# EPICS IOC start-up script: iocBoot/common/startup.RK_CA3900.iocsh
# IOC shell script for R&K CA3900 SSA
# Includes modbus config and db loading
# Required macros:
# PORT - asyn port
# P - PV name prefix
# IP - IP address or host name

# Use the following commands for TCP/IP
# drvAsynIPPortConfigure(const char *portName, const char *hostInfo,
# 			 unsigned int priority, int noAutoConnect,
#			 int noProcessEos);

drvAsynIPPortConfigure("$(PORT)", "$(IP):502", 0,0,1)
dbLoadRecords("db/asynRecord.db","P=$(P), R=ASYN, PORT=$(PORT), ADDR=0,IMAX=0,OMAX=0")

# modbusInterposeConfig(const char *portName, modbusLinkType linkType,
#			int timeoutMsec, int writeDelayMsec)
# linkType 0 = TCP/IP
modbusInterposeConfig("$(PORT)", 0, 1500, 0)

# Modbus function code: 3 (Read Holding Registers, 16-bit word access)
# Start address: 1
# Access 125 words as inputs
# Default data type: unsigned integer
# drvModbusAsynConfigure("portName", "TcpPortName", slaveaddress,
#			modbusFunctions, modbusStartAddress, modbusLength,
#			dataType, pollMsec, "plcType")
#
drvModbusAsynConfigure("$(PORT)_inw1", "$(PORT)", 0, 3, 1, 125, 0, 500, "RK")
dbLoadRecords("db/asynRecord.db", "P=$(P), R=ASYN_IN, PORT=$(PORT)_inw1, ADDR=0,IMAX=0,OMAX=0")
dbLoadRecords("db/statistics.template", "P=$(P), R=ASYN_IN, PORT=$(PORT)_inw1, SCAN=10 second")

# Modbus function code: 3 (Read Holding Registers, 16-bit word access)
# Start address: 125
# Access 16 words as inputs
# Default data type: unsigned integer
drvModbusAsynConfigure("$(PORT)_inw2", "$(PORT)", 0, 3, 125, 16, 0, 5000, "RK")
dbLoadRecords("db/asynRecord.db", "P=$(P), R=ASYN_IN, PORT=$(PORT)_inw2, ADDR=0,IMAX=0,OMAX=0")

# Modbus function code: 3 (Read Holding Registers, 16-bit word access)
# Start address: 171
# Access 20 words as inputs
# Default data type: unsigned integer
drvModbusAsynConfigure("$(PORT)_inw3", "$(PORT)", 0, 3, 171, 20, 0, 5000, "RK")
dbLoadRecords("db/asynRecord.db", "P=$(P), R=ASYN_IN, PORT=$(PORT)_inw3, ADDR=0,IMAX=0,OMAX=0")

# Modbus function code: 6 (Write Single Register, 16-bit word access)
# Start address: 1
# Access 7 words as outputs
# Default data type: unsigned integer
drvModbusAsynConfigure("$(PORT)_outw1", "$(PORT)", 0, 6, 1, 7, 0, 100, "RK")
dbLoadRecords("db/asynRecord.db","P=$(P), R=ASYN_OUT, PORT=$(PORT)_outw1, ADDR=0,IMAX=0,OMAX=0")
dbLoadRecords("db/statistics.template", "P=$(P), R=ASYN_OUT, PORT=$(PORT)_outw1, SCAN=10 second")

# Modbus function code: 6 (Write Single Register, 16-bit word access)
# Start address: 128
# Access 5 words as outputs
# Default data type: unsigned integer
drvModbusAsynConfigure("$(PORT)_outw2", "$(PORT)", 0, 6, 128, 5, 0, 100, "RK")
dbLoadRecords("db/asynRecord.db","P=$(P), R=ASYN_OUT, PORT=$(PORT)_outw2, ADDR=0,IMAX=0,OMAX=0")

# Enable ASYN_TRACEIO_HEX on octet server
asynSetTraceIOMask("$(PORT)", 0, 0x4)
# Enable ASYN_TRACE_ERROR and ASYN_TRACEIO_DRIVER on octet server
#asynSetTraceMask("$(PORT)", 0, 0x9)
# Dump up to 256 bytes in asynTrace
asynSetTraceIOTruncateSize("$(PORT)", 0, 256)

# Enable ASYN_TRACEIO_HEX on modbus server
asynSetTraceIOMask("$(PORT)_inw1", 0, 0x4)
asynSetTraceIOMask("$(PORT)_inw2", 0, 0x4)
asynSetTraceIOMask("$(PORT)_inw3", 0, 0x4)
# Enable ASYN_TRACE_FLOW on modbus server
#asynSetTraceMask("$(PORT)_inw1", 0, 0x11)
#asynSetTraceMask("$(PORT)_inw2", 0, 0x11)
#asynSetTraceMask("$(PORT)_inw3", 0, 0x11)
# Dump up to 512 bytes in asynTrace
asynSetTraceIOTruncateSize("$(PORT)_inw1", 0, 512)
asynSetTraceIOTruncateSize("$(PORT)_inw2", 0, 512)
asynSetTraceIOTruncateSize("$(PORT)_inw3", 0, 512)

# Load records
dbLoadRecords("db/ssa_RK_CA3900.db", "P=$(P),CAV1=$(CAV1=None),CAV2=$(CAV2=None),PORT_P=$(PORT),ASG=$(ASG)")

# Just in case
epicsThreadSleep(0.25)

# End of script
